_CFC_ (* Continuous Function Chart, elements in execution order *)
#0 MUX(#6, 0, SIZEOF(RD_1), SIZEOF(RD_2), SIZEOF(RD_3))
#1 OR(SHU6_PV1_UST_RE_PUSK, SHU6_PV1_UST_RE_RABOTA)
#2 TON1:TON(IN: NOT #7.out 1, PT: T#500ms)
#3 RT_ModBus:R_TRIG(CLK: #2.Q)
#4 CTU_ModBus:CTU(CU: #3.Q, RESET: #4.Q, PV: 2)
#5 ADD(#4.CV, 1)
#6 WORD_TO_BYTE(#5)
#7 MB_READ_REGS:ModbusRtuMaster_KL6x22B.ReadRegs(#6, Quantity, MBAddr, #0, #15, #20.Q, T#1s)
#8 Errorld <= #7.out 3
#9 cbRead <= #7.out 4
#10 AND(#12, #7.out 2, #1)
#11 SHU6_PV1_MP1_OBR_ERROR <= #10
#12 =(1, #6)
#13 AND(#18, #7.out 2, #1)
#14 SHU6_PV1_MV1_OBR_ERROR <= #13
#15 MUX(#6, 0, ADR(RD_1), ADR(RD_2), ADR(RD_3))
#16 AND(#19, #7.out 2, #1)
#17 SHU6_PV1_MRQ1_OBR_ERROR <= #16
#18 =(2, #6)
#19 =(3, #6)
#20 TON2:TON(IN: #2.Q, PT: T#500ms)
_END_CFC_
END_PROGRAM
